# EPICS StreamDevice protocol: protocols/signal.proto
Terminator = LF;
ExtraInput = Ignore;

setSig {
	out "\$1=%(A)d,%(B)d,%(C)d";
}

getSig {
	out "\$1";
	in "\$1=%d,%*d,%*d";
	@replytimeout {
		disconnect;
		wait 2000;
		connect 1000;
	}
}

getSigDx {
	in "\$1=%*d,%d,%*d";
}

getSigSense {
	in "\$1=%*d,%*d,%d";
}
